Staubli VAL3: link_all.pgx

public program link_all(string x_sName)
  local num i
begin
  // link all
  link(tTraj[x_sName].fReference,world)
  tTraj[x_sName].fReference.trsf=saveData:fFrameItem[tTraj[x_sName].nIndexFrame].fFrame.trsf
  link(tTraj[x_sName].fFrame,tTraj[x_sName].fReference)
  link(tTraj[x_sName].pO,tTraj[x_sName].fReference)
  link(tTraj[x_sName].pX,tTraj[x_sName].fReference)
  link(tTraj[x_sName].pY,tTraj[x_sName].fReference)
  link(tTraj[x_sName].pZ,tTraj[x_sName].fReference)
  for i=0 to size(tTraj[x_sName].tData)-1
    link(tTraj[x_sName].tData[i].pPoint,tTraj[x_sName].fFrame)
  endFor
end
